FUNCTION_BLOCK AddMoverToGroupTask EXTENDS TaskBase
VAR_INPUT
END_VAR
VAR_OUTPUT
END_VAR
VAR
	AddtoGrp			: MC_AddAxisToGroup;
	_CaGroup			: ICollisionGroup;
	_Axis				: REFERENCE TO AXIS_REF;
	_addMover : BOOL;
	_moverNumber : UDINT;
END_VAR

{analysis -2}

METHOD Abort : BOOL
AddtoGrp.Execute := FALSE;
Abort := true;
State := 0;
END_METHOD

METHOD AddMover : BOOL
VAR_INPUT
	MoverToAdd : I_XtsMoverAxis;
END_VAR
_Axis REF= MoverToAdd.AxisRef;
AddtoGrp.IdentInGroup := MoverToAdd.IdentInGroup;
_Busy := TRUE;
AddMover := _addMover := TRUE;
END_METHOD

METHOD Cycle : HRESULT
VAR_INPUT
END_VAR
Cycle := S_OK;
CASE State OF
	0:
		IF _addMover THEN
			Cycle := S_PENDING;
			_Done := FALSE;
			_Error := FALSE;
			_Busy := TRUE;
			AddtoGrp.Execute := TRUE;
			IF AddtoGrp.Busy THEN
				State := 10;
				_addMover := FALSE;
			END_IF
		END_IF
	
	10:
		IF NOT AddtoGrp.Busy THEN
			IF AddtoGrp.Done THEN
				_Done := TRUE;
			ELSIF AddtoGrp.Error THEN
				_Error := TRUE;
			END_IF
			_Busy := FALSE;
			AddtoGrp.Execute := false;
			State := 0;
			Cycle := S_OK;
		END_IF
	ELSE
		Cycle := E_FAIL;
END_CASE

AddtoGrp(AxesGroup := _CaGroup.GroupRef,
			Axis := _Axis);
END_METHOD

METHOD FB_init : BOOL
VAR_INPUT
	bInitRetains : BOOL; // if TRUE, the retain variables are initialized (warm start / cold start)
	bInCopyCode : BOOL;  // if TRUE, the instance afterwards gets moved into the copy code (online change)
	myCaGroup : ICollisionGroup;	
END_VAR
_CaGroup := myCaGroup;
END_METHOD

END_FUNCTION_BLOCK

(* stored: Version 1.1.0.1, ProductVersion 3.1.4024.12
   POU AddMoverToGroupTask: Id {8561ba4a-bbc2-4a4c-8d8e-313f70a4cd47}, SpecialFunc None
   Method Abort: Id {f17ab960-5dcf-47aa-8c4d-ce7d93fe1bb1}
   Method AddMover: Id {481f5339-50ec-48c8-9b4c-100ecb265f94}
   Method Cycle: Id {6096abf8-fe4d-4db3-982a-c3405f3d7073}
   Method FB_init: Id {1a3771d2-cfdd-44cb-ac56-4c890f762040} *)
